// TIA Portal V20 export
TYPE "Udt_M200D_IN"
   STRUCT
      "Ready (automatic)" : Bool;
      "Motor on" : Bool;
      "Group fault" : Bool;
      "Group warning" : Bool;
      "Input 1_Stop" : Bool;
      "Input 2_Ocuupy" : Bool;
      "Input 3" : Bool;
      "Input 4" : Bool;
      "Current motor current Icurr % Bit 0" : Bool;
      "Current motor current Icurr % Bit 1" : Bool;
      "Current motor current Icurr % Bit 2" : Bool;
      "Current motor current Icurr % Bit 3" : Bool;
      "Current motor current Icurr % Bit 4" : Bool;
      "Current motor current Icurr % Bit 5" : Bool;
      "Manual mode local mode" : Bool;
      "Ramp operation" : Bool;
   END_STRUCT;
END_TYPE
